FUNCTION_BLOCK PUBLIC ShutDown
VAR_INPUT
	GvlIdentifier : STRING;
END_VAR
VAR_OUTPUT
END_VAR
VAR
END_VAR

IF GvlIdentifier = 'R1' THEN
	R1.RecipeStatus := FALSE;
	R1.HeatCoolStatus := FALSE;
	R1.StirrerStatus := FALSE;
	R1.AbortRecipe := FALSE;
	R1.DosingPumpStatus :=FALSE;
END_IF

END_FUNCTION_BLOCK

(* stored: Version 1.1.0.1, ProductVersion 3.1.4024.3
   POU ShutDown: Id {2fd1b10f-dd9e-4f28-922f-b0db218af6ba}, SpecialFunc None *)
